// TIA Portal V20 export
TYPE "typeEm2Commands"
// stored: Access Published, Namespace Unit1
   STRUCT
      jobinterface { ExternalWritable := 'False'} : "Unit1.typeEm2CommandsJobInterface";
   END_STRUCT;
END_TYPE
